{attribute 'linkalways'} 
{attribute 'no_explicit_call' := 'This FB is a CLASS and must be accessed using methods or properties'}
{attribute 'enable_dynamic_creation'}
FUNCTION_BLOCK PlcNodePack
VAR
    // Conversion
	// DINT_TO
	node_DINT_TO_LREAL : Node_DINT_TO_LREAL;
	node_DINT_TO_REAL : Node_DINT_TO_REAL;
	// LREAL_TO_
	node_LREAL_TO_DINT : Node_LREAL_TO_DINT;
	node_LREAL_TO_UDINT : Node_LREAL_TO_UDINT;
	// REAL_TO_
    node_REAL_TO_DINT : Node_REAL_TO_DINT;
	node_REAL_TO_UDINT : Node_REAL_TO_UDINT;
	// UDINT_TO
	node_UDINT_TO_LREAL : Node_UDINT_TO_LREAL;
	node_UDINT_TO_REAL : Node_UDINT_TO_REAL;
    // Logic
    node_NOT : Node_NOT;
    node_AND : Node_AND;
    node_NAND : Node_NAND;
    node_OR : Node_OR;
    node_NOR : Node_NOR;
    node_XOR : Node_XOR;
    node_XNOR : Node_XNOR;
	
	// TwinCAT
	node_TwinCATStatus : Node_TwinCATStatus;
	
	// Strings
	node_CONCAT : Node_CONCAT;
    node_DELETE : Node_DELETE;
    node_FIND : Node_FIND;
    node_INSERT : Node_INSERT;
    node_LEFT : Node_LEFT;
    node_LEN : Node_LEN;
    node_MID : Node_MID;
	node_REPLACE : Node_REPLACE;
    node_RIGHT : Node_RIGHT;
	
END_VAR

METHOD PUBLIC RegisterWithNodeFactory
VAR_INPUT
	NodeFactory : I_NodeFactory;
END_VAR
// Conversion
NodeFactory.AddNodeAsPrototype('PLC/Convert/DINT/DINT_TO_LREAL', node_DINT_TO_LREAL);
NodeFactory.AddNodeAsPrototype('PLC/Convert/DINT/DINT_TO_REAL', node_DINT_TO_REAL);
NodeFactory.AddNodeAsPrototype('PLC/Convert/LREAL/LREAL_TO_DINT', node_LREAL_TO_DINT);
NodeFactory.AddNodeAsPrototype('PLC/Convert/LREAL/LREAL_TO_UDINT', node_LREAL_TO_UDINT);
NodeFactory.AddNodeAsPrototype('PLC/Convert/REAL/REAL_TO_DINT', node_REAL_TO_DINT);
NodeFactory.AddNodeAsPrototype('PLC/Convert/REAL/REAL_TO_UDINT', node_REAL_TO_UDINT);
NodeFactory.AddNodeAsPrototype('PLC/Convert/UDINT/UDINT_TO_LREAL', node_UDINT_TO_LREAL);
NodeFactory.AddNodeAsPrototype('PLC/Convert/UDINT/UDINT_TO_REAL', node_UDINT_TO_REAL);

// Logic
NodeFactory.AddNodeAsPrototype('PLC/Logic/NOT', node_NOT);
NodeFactory.AddNodeAsPrototype('PLC/Logic/AND', node_AND);
NodeFactory.AddNodeAsPrototype('PLC/Logic/NAND', node_NAND);
NodeFactory.AddNodeAsPrototype('PLC/Logic/OR', node_OR);
NodeFactory.AddNodeAsPrototype('PLC/Logic/NOR', node_NOR);
NodeFactory.AddNodeAsPrototype('PLC/Logic/XOR', node_XOR);
NodeFactory.AddNodeAsPrototype('PLC/Logic/XNOR', node_XNOR);

// Hardware
//NodeFactory.AddNodeAsPrototype('PLC/Hardware/DI', node_DigitalInput);
//NodeFactory.AddNodeAsPrototype('PLC/Hardware/DO', node_DigitalOutput);

// TwinCAT
//NodeFactory.AddNodeAsPrototype('PLC/TwinCAT/TwinCAT Status', node_TwinCATStatus);

// Strings
NodeFactory.AddNodeAsPrototype('PLC/Strings/CONCAT', node_CONCAT);
NodeFactory.AddNodeAsPrototype('PLC/Strings/DELETE', node_DELETE);
NodeFactory.AddNodeAsPrototype('PLC/Strings/FIND', node_FIND);
NodeFactory.AddNodeAsPrototype('PLC/Strings/INSERT', node_INSERT);
NodeFactory.AddNodeAsPrototype('PLC/Strings/LEFT', node_LEFT);
NodeFactory.AddNodeAsPrototype('PLC/Strings/LEN', node_LEN);
NodeFactory.AddNodeAsPrototype('PLC/Strings/MID', node_MID);
NodeFactory.AddNodeAsPrototype('PLC/Strings/REPLACE', node_REPLACE);
NodeFactory.AddNodeAsPrototype('PLC/Strings/RIGHT', node_RIGHT);
END_METHOD

END_FUNCTION_BLOCK

(* stored: Version 1.1.0.1, ProductVersion 3.1.4026.18
   POU PlcNodePack: Id {257fc325-f932-4b89-a50a-e9a0a38418f4}, SpecialFunc None
   Method RegisterWithNodeFactory: Id {9eda346d-cc38-44e9-a636-4948bc24f687} *)
